{attribute addProperty BoxType "EL3632-0000-0016"}
{attribute addProperty Id "Ch1_StatusAT %I*Ch1_Status_15B44ED31620Ch1_SampleAT %I*ARRAY[0..9] OF Ch1_Sample_37C07C83160200Ch2_StatusAT %I*Ch2_Status_15B44ED31620Ch2_SampleAT %I*ARRAY[0..9] OF Ch2_Sample_29ECE468160200Next_Sync1_TimeAT %I*Next_Sync1_Time_F650E6AF6480Sample_CountAT %I*Sample_Count_7FA7B6EB1620WcStateAT %I*WcState_98A4DF7520.250InfoDataAT %I*InfoData_0BDED7BF144180"}
{attribute addProperty CRC "3939910614"}
{attribute addProperty SizeInBites "578"}
{attribute addProperty SizeInBytes "72.25"}
TYPE EL3632_D178097B :
STRUCT
	{attribute addProperty Name "Ch1_Status"}
	Ch1_Status : Ch1_Status_15B44ED3;
	{attribute addProperty Name "Ch1_Sample"}
	Ch1_Sample : ARRAY[0..9] OF Ch1_Sample_37C07C83;
	{attribute addProperty Name "Ch2_Status"}
	Ch2_Status : Ch2_Status_15B44ED3;
	{attribute addProperty Name "Ch2_Sample"}
	Ch2_Sample : ARRAY[0..9] OF Ch2_Sample_29ECE468;
	{attribute addProperty Name "Next_Sync1_Time"}
	Next_Sync1_Time : Next_Sync1_Time_F650E6AF;
	{attribute addProperty Name "Sample_Count"}
	Sample_Count : Sample_Count_7FA7B6EB;
	{attribute addProperty Name "WcState"}
	WcState : WcState_98A4DF75;
	{attribute addProperty Name "InfoData"}
	InfoData : InfoData_0BDED7BF;
END_STRUCT
END_TYPE

(* stored: Version 1.2.0.0, ProductVersion 3.1.4024.9
   DUT EL3632_D178097B: Id {134cb78e-d788-48ca-95d2-5ce023287f9e} *)
